(* IEC 61131-3 sources: Test002/ConveyorBelt/Class/ConveyorBelt, 1 file *)

(* ---- ConveyorBelt.st ---- *)
(*!
<Class
	Name               = "ConveyorBelt"
	Revision           = "1.0"
	RealtimeTask       = "false"
	CyclicTask         = "true"
	DefCyclictime      = "10 ms"
	BackgroundTask     = "false"
	Sigmatek           = "false"
	OSInterface        = "false"
	HighPriority       = "false"
	Automatic          = "false"
	UpdateMode         = "Prescan"
	SharedCommandTable = "true"
	Objectsize         = "(284,120)">
	<Channels>
		<Server Name="ClassSvr" Visualized="false" Initialize="false" WriteProtected="true" Retentive="false"/>
		<Server Name="ConveyorbeltSteps" Visualized="false" Initialize="true" DefValue="Step01" WriteProtected="false" Retentive="false"/>
		<Server Name="TimeDelay" Visualized="false" Initialize="true" DefValue="2000" WriteProtected="false" Retentive="File"/>
		<Client Name="Cylinder" Required="true" Internal="false"/>
		<Client Name="Lichtschrank" Required="true" Internal="false"/>
		<Client Name="Motor" Required="true" Internal="false"/>
		<Client Name="Start" Required="true" Internal="false"/>
	</Channels>
</Class>
*)
ConveyorBelt : CLASS
	TYPE
	  t_ConveyorSteps :  //! <Type Public="true" Name="t_ConveyorSteps"/>
	  (
	    Step01:=1,
	    Step02:=2,
	    Step03:=3,
	    Step04:=4
	  )$UDINT;
	END_TYPE
  //Servers:
	ClassSvr 	: SvrChCmd_DINT;
	TimeDelay 	: SvrCh_UDINT;
	ConveyorbeltSteps 	: SvrCh_t_ConveyorSteps_PTofCls_ConveyorBelt;
  //Clients:
	Motor 	: CltCh_DINT;
	Lichtschrank 	: CltCh_DINT;
	Start 	: CltCh_DINT;
	Cylinder 	: CltCh_DINT;
  //Variables:
		TimeMark 	: UDINT;
  //Functions:

	FUNCTION VIRTUAL GLOBAL CyWork
		VAR_INPUT
			EAX 	: UDINT;
		END_VAR
		VAR_OUTPUT
			state (EAX) 	: UDINT;
		END_VAR;
  //Tables:
	FUNCTION @STD
		VAR_OUTPUT
			ret_code	: CONFSTATES;
		END_VAR;
	FUNCTION GLOBAL TAB @CT_;
END_CLASS;

FUNCTION VIRTUAL GLOBAL ConveyorBelt::CyWork
	VAR_INPUT
		EAX 	: UDINT;
	END_VAR
	VAR_OUTPUT
		state (EAX) 	: UDINT;
	END_VAR
  VAR
  	vergangenZeit : UDINT;
    vergangenZeitQ : BOOL;
  END_VAR

  Lichtschrank := Lichtschrank.Read();
  Start := Start.Read();

  //Vergangenzeit

  if TimeMark > 0 then
    vergangenZeit := (ops.tAbsolute - TimeMark);
    vergangenZeitQ := vergangenZeit > TimeDelay;
  else
    vergangenZeit := 0;
  end_if;

  case ConveyorbeltSteps of
  	ConveyorBelt::t_ConveyorSteps::Step01:  //Start Conveyor

 //*************Step 01******************\\
      if(Start = 1 AND Lichtschrank = 1) then

        Motor := 1;
        Cylinder := 0;

        TimeMark := ops.tAbsolute;
        ConveyorbeltSteps := Step02;

      elsif(Start = 1 and Lichtschrank = 0) then //Warte auf frei Lichtschrank

        Motor := 0;
        Cylinder := 0;

      end_if;

//*************Step 02******************\\

  	ConveyorBelt::t_ConveyorSteps::Step02:   //Warte auf Zeit

        if vergangenZeitQ then

          Cylinder := 1;
          Motor := 0;
          TimeMark := 0;
          ConveyorbeltSteps := Step03;
        end_if;

 //*************Step 03******************\\
  	ConveyorBelt::t_ConveyorSteps::Step03:

        if Start = 1 and Lichtschrank = 0 then

          Cylinder := 1;
          Motor := 0;
          TimeMark := ops.tAbsolute;
          ConveyorbeltSteps := Step04;

        end_if;

        IF Lichtschrank and Lichtschrank = 0 THEN

          Lichtschrank := 0;
        END_IF;

//*************Step 04******************\\

  	ConveyorBelt::t_ConveyorSteps::Step04:

        if Start = 0  and vergangenZeitQ then

          Cylinder := 0;
          Motor := 0;
          TimeMark := 0;
          ConveyorbeltSteps := Step01;

        end_if;

  end_case;

  Motor.Write (Motor);
  Cylinder.Write (Cylinder);

	state := READY;

END_FUNCTION
